FUNCTION_BLOCK DoorControl (* Basic Function Block Type *)
  (* Standard: 61499-2 *)
  (* Version 0.0, 6/17/2016, Andrei, nxtControl GmbH, Template *)
  PACKAGE Main;
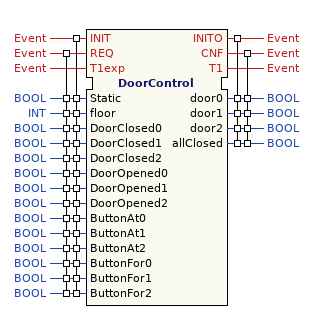
  EVENT_INPUT
    INIT WITH Static, floor, DoorClosed0, DoorClosed1, DoorClosed2, DoorOpened0, DoorOpened1, DoorOpened2, ButtonAt0, ButtonAt1, ButtonAt2, ButtonFor0, ButtonFor1, ButtonFor2; (* Initialization Request *)
    REQ WITH Static, floor, DoorClosed0, DoorClosed1, DoorClosed2, DoorOpened0, DoorOpened1, DoorOpened2, ButtonAt0, ButtonAt1, ButtonAt2, ButtonFor0, ButtonFor1, ButtonFor2; (* Normal Execution Request *)
    T1exp;
  END_EVENT
  EVENT_OUTPUT
    INITO WITH door0, door1, door2, allClosed; (* Initialization Confirm *)
    CNF WITH door0, door1, door2, allClosed; (* Execution Confirmation *)
    T1;
  END_EVENT
  VAR_INPUT
    Static : BOOL;
    floor : INT;
    DoorClosed0 : BOOL;
    DoorClosed1 : BOOL;
    DoorClosed2 : BOOL;
    DoorOpened0 : BOOL;
    DoorOpened1 : BOOL;
    DoorOpened2 : BOOL;
    ButtonAt0 : BOOL;
    ButtonAt1 : BOOL;
    ButtonAt2 : BOOL;
    ButtonFor0 : BOOL;
    ButtonFor1 : BOOL;
    ButtonFor2 : BOOL;
  END_VAR
  VAR_OUTPUT
    door0 : BOOL;
    door1 : BOOL;
    door2 : BOOL;
    allClosed : BOOL;
  END_VAR
  VAR
    doOpen0 : BOOL;
    doOpen1 : BOOL;
    doOpen2 : BOOL;
  END_VAR
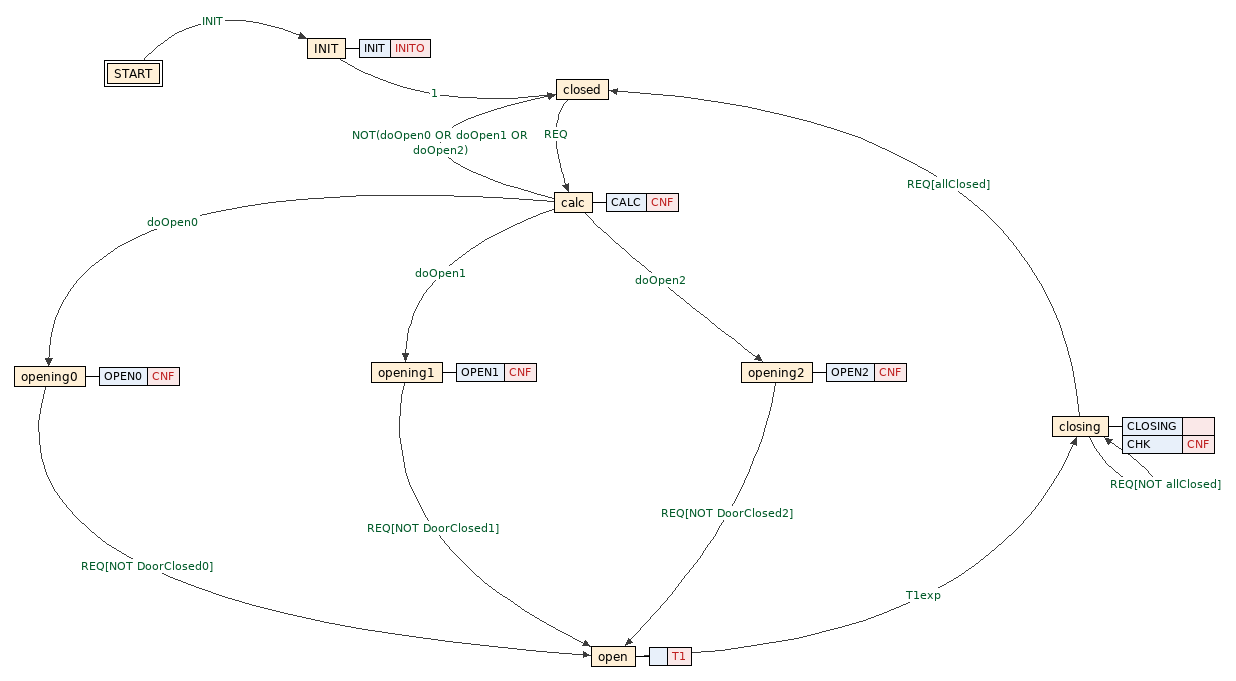
  EC_STATES
    START; (* Initial State *)
    INIT : INIT -> INITO;
    closed;
    open : -> T1;
    closing : CLOSING, CHK -> CNF;
    opening0 : OPEN0 -> CNF;
    opening1 : OPEN1 -> CNF;
    opening2 : OPEN2 -> CNF;
    calc : CALC -> CNF;
  END_STATES
  EC_TRANSITIONS
    START TO INIT := INIT;
    INIT TO closed := 1;
    opening0 TO open := REQ[NOT DoorClosed0];
    opening1 TO open := REQ[NOT DoorClosed1];
    opening2 TO open := REQ[NOT DoorClosed2];
    calc TO opening0 := doOpen0;
    calc TO opening1 := doOpen1;
    calc TO opening2 := doOpen2;
    open TO closing := T1exp;
    closed TO calc := REQ;
    closing TO closed := REQ[allClosed];
    closing TO closing := REQ[NOT allClosed];
    calc TO closed := NOT(doOpen0 OR doOpen1 OR doOpen2);
  END_TRANSITIONS
  ALGORITHM INIT IN ST: (* Initialization algorithm *)
;
allClosed:=DoorClosed0 & DoorClosed1 & DoorClosed2;
  END_ALGORITHM
  ALGORITHM CALC IN ST:
doOpen0:=(floor=0) AND (ButtonAt0 OR ButtonFor0);
doOpen1:=(floor=1) AND (ButtonAt1 OR ButtonFor1);
doOpen2:=(floor=2) AND (ButtonAt2 OR ButtonFor2);

allClosed:=DoorClosed0 & DoorClosed1 & DoorClosed2;
  END_ALGORITHM
  ALGORITHM CHK IN ST:
allClosed:=DoorClosed0 & DoorClosed1 & DoorClosed2;
  END_ALGORITHM
  ALGORITHM OPEN0 IN ST:
door0:=TRUE;
  END_ALGORITHM
  ALGORITHM OPEN1 IN ST:
door1:=TRUE;;
  END_ALGORITHM
  ALGORITHM OPEN2 IN ST:
door2:=TRUE;
  END_ALGORITHM
  ALGORITHM CLOSING IN ST:
door0:=FALSE;
door1:=FALSE;
door2:=FALSE;
  END_ALGORITHM
END_FUNCTION_BLOCK
